% RSLogix 500 project DRUCKREGELUNG MIT PUMPE UND SIGNALANZEIGE.RSS, saved by version 8.30.00.16 %
PROJECT "UNTITLED"    % processor: Bul.1763 MicroLogix 1100 Series B %

PROGRAM FILES
  LAD 2 "MAIN"  3 rungs
  LAD 3 "DIGITAL IO"  5 rungs
  LAD 4 "CONTROLS"  11 rungs

DATA FILES
  O0 OUTPUT  4 elements
  I1 INPUT  6 elements
  S2 STATUS  66 elements
  B3 BINARY  1 elements
  T4 TIMER  4 elements
  C5 COUNTER  1 elements
  R6 CONTROL  1 elements
  N7 INTEGER  2 elements
  F8 FLOAT  1 elements

LADDER 2 "MAIN"
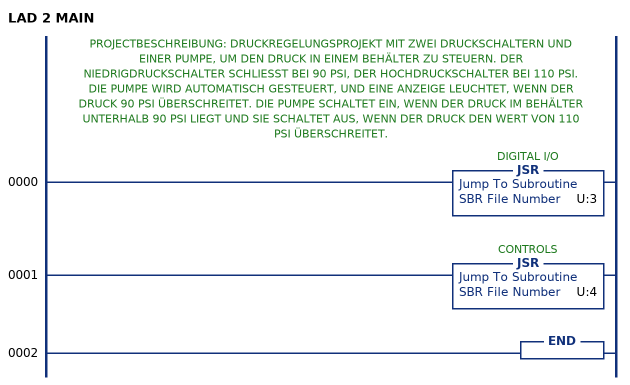
% Rung: 0 %
% PROJECTBESCHREIBUNG: DRUCKREGELUNGSPROJEKT MIT ZWEI DRUCKSCHALTERN UND EINER PUMPE, UM DEN DRUCK IN EINEM BEHÄLTER ZU STEUERN. DER NIEDRIGDRUCKSCHALTER SCHLIESST BEI 90 PSI, DER HOCHDRUCKSCHALTER BEI 110 PSI. DIE PUMPE WIRD AUTOMATISCH GESTEUERT, UND EINE ANZEIGE LEUCHTET, WENN DER DRUCK 90 PSI ÜBERSCHREITET. DIE PUMPE SCHALTET EIN, WENN DER DRUCK IM BEHÄLTER UNTERHALB 90 PSI LIEGT UND SIE SCHALTET AUS, WENN DER DRUCK DEN WERT VON 110 PSI ÜBERSCHREITET. %
SOR JSR U:3 EOR
%   U:3  "DIGITAL I/O" %
% Rung: 1 %
SOR JSR U:4 EOR
%   U:4  "CONTROLS" %
% Rung: 2 %
SOR END EOR

LADDER 3 "DIGITAL IO"
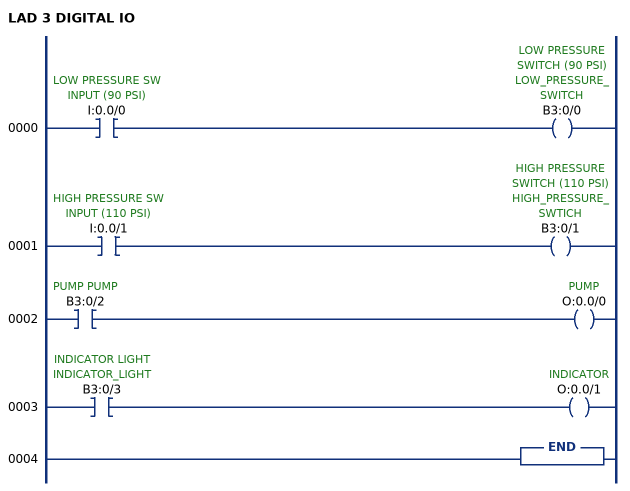
% Rung: 0 %
SOR XIC I:0.0/0 OTE B3:0/0 EOR
%   I:0.0/0  "LOW PRESSURE SW INPUT (90 PSI)" %
%   B3:0/0  LOW_PRESSURE_SWITCH  "LOW PRESSURE SWITCH (90 PSI)" %
% Rung: 1 %
SOR XIC I:0.0/1 OTE B3:0/1 EOR
%   I:0.0/1  "HIGH PRESSURE SW INPUT (110 PSI)" %
%   B3:0/1  HIGH_PRESSURE_SWTICH  "HIGH PRESSURE SWITCH (110 PSI)" %
% Rung: 2 %
SOR XIC B3:0/2 OTE O:0.0/0 EOR
%   B3:0/2  PUMP  "PUMP" %
%   O:0.0/0  "PUMP" %
% Rung: 3 %
SOR XIC B3:0/3 OTE O:0.0/1 EOR
%   B3:0/3  INDICATOR_LIGHT  "INDICATOR LIGHT" %
%   O:0.0/1  "INDICATOR" %
% Rung: 4 %
SOR END EOR

LADDER 4 "CONTROLS"
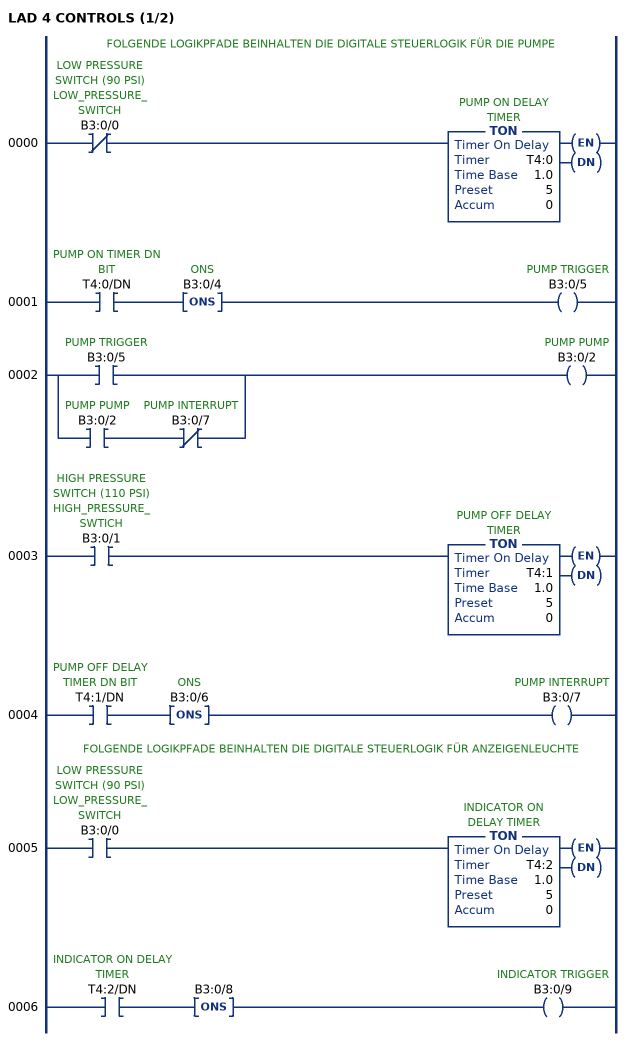
% Rung: 0 %
% FOLGENDE LOGIKPFADE BEINHALTEN DIE DIGITALE STEUERLOGIK FÜR DIE PUMPE %
SOR XIO B3:0/0 TON T4:0 1.0 5 0 EOR
%   B3:0/0  LOW_PRESSURE_SWITCH  "LOW PRESSURE SWITCH (90 PSI)" %
%   T4:0  "PUMP ON DELAY TIMER" %
% Rung: 1 %
SOR XIC T4:0/DN ONS B3:0/4 OTE B3:0/5 EOR
%   T4:0/DN  "PUMP ON TIMER DN BIT" %
%   B3:0/4  "ONS" %
%   B3:0/5  "PUMP TRIGGER" %
% Rung: 2 %
SOR BST XIC B3:0/5 NXB XIC B3:0/2 XIO B3:0/7 BND OTE B3:0/2 EOR
%   B3:0/5  "PUMP TRIGGER" %
%   B3:0/2  PUMP  "PUMP" %
%   B3:0/7  "PUMP INTERRUPT" %
% Rung: 3 %
SOR XIC B3:0/1 TON T4:1 1.0 5 0 EOR
%   B3:0/1  HIGH_PRESSURE_SWTICH  "HIGH PRESSURE SWITCH (110 PSI)" %
%   T4:1  "PUMP OFF DELAY TIMER" %
% Rung: 4 %
SOR XIC T4:1/DN ONS B3:0/6 OTE B3:0/7 EOR
%   T4:1/DN  "PUMP OFF DELAY TIMER DN BIT" %
%   B3:0/6  "ONS" %
%   B3:0/7  "PUMP INTERRUPT" %
% Rung: 5 %
% FOLGENDE LOGIKPFADE BEINHALTEN DIE DIGITALE STEUERLOGIK FÜR ANZEIGENLEUCHTE %
SOR XIC B3:0/0 TON T4:2 1.0 5 0 EOR
%   B3:0/0  LOW_PRESSURE_SWITCH  "LOW PRESSURE SWITCH (90 PSI)" %
%   T4:2  "INDICATOR ON DELAY TIMER" %
% Rung: 6 %
SOR XIC T4:2/DN ONS B3:0/8 OTE B3:0/9 EOR
%   T4:2  "INDICATOR ON DELAY TIMER" %
%   B3:0/9  "INDICATOR TRIGGER" %

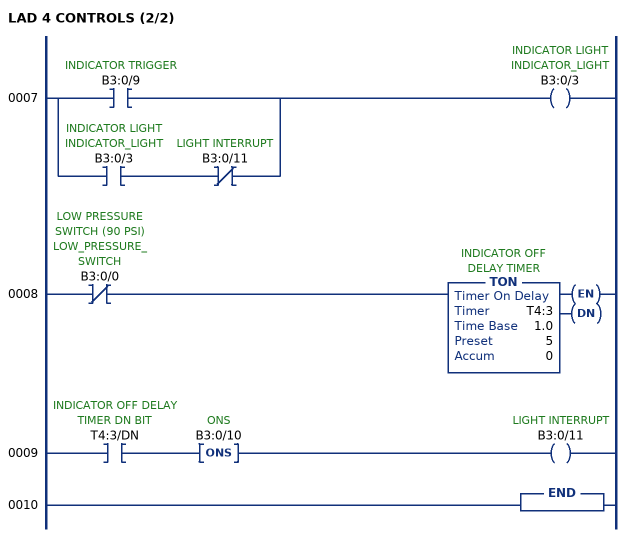
% Rung: 7 %
SOR BST XIC B3:0/9 NXB XIC B3:0/3 XIO B3:0/11 BND OTE B3:0/3 EOR
%   B3:0/9  "INDICATOR TRIGGER" %
%   B3:0/3  INDICATOR_LIGHT  "INDICATOR LIGHT" %
%   B3:0/11  "LIGHT INTERRUPT" %
% Rung: 8 %
SOR XIO B3:0/0 TON T4:3 1.0 5 0 EOR
%   B3:0/0  LOW_PRESSURE_SWITCH  "LOW PRESSURE SWITCH (90 PSI)" %
%   T4:3  "INDICATOR OFF DELAY TIMER" %
% Rung: 9 %
SOR XIC T4:3/DN ONS B3:0/10 OTE B3:0/11 EOR
%   T4:3/DN  "INDICATOR OFF DELAY TIMER DN BIT" %
%   B3:0/10  "ONS" %
%   B3:0/11  "LIGHT INTERRUPT" %
% Rung: 10 %
SOR END EOR

OTHER DOCUMENTED ADDRESSES
  I:1.0/0  "LOW PRESSURE SWITCH INPUT"
  I:1.0/1  "HIGH PRESSURE SWITCH INPUT"
  N7:0  "RUNNING MODES 1) L & H OFF 2) L ON & H OFF INI 3) L & H ON 4) L ON & H TURN OFF"
  N7:1  "LAST MODE"
  O:2.0/0  "PUMP OUTPUT"
  O:2.0/1  "INDICATOR LIGHT"
  U:5  "CONTROLS"
  U:6  "PUMP"

DATA TABLE (non-zero values as saved)
DATA B3
% B3:0 % 0X0024
DATA T4
% .PRE .ACC %
% T4:0 % 5 0
% T4:1 % 5 0
% T4:2 % 5 0
% T4:3 % 5 0
DATA N7
% N7:0 % 1 0
